// TIA Portal V20 export
TYPE "typeSequenceControlNodeHomeCheck_sideTapeAttachment"
// stored: Namespace Unit1.Em4
   STRUCT
      waitPosTapeGetReq { ExternalWritable := 'False'} : Bool;
      waitPosTapeLeftGet { ExternalWritable := 'False'} : Bool;
      waitPosTapeRightGet { ExternalWritable := 'False'} : Bool;
      waitPosTapeAllGet { ExternalWritable := 'False'} : Bool;
      putPosTapeAllGet { ExternalWritable := 'False'} : Bool;
   END_STRUCT;
END_TYPE
